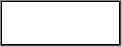
VISUALIZATION VISU_SubSystemButton  // 122x47
VAR_IN_OUT
    widget : SubSystemButtonWidget;
END_VAR
    Rectangle (0,0 120x45), invisible if: widget.isNotOrange
    Rectangle (0,0 120x45), invisible if: widget.isNotGray
    Rectangle (0,0 120x45), invisible if: widget.isNotBlue
    Rectangle (0,0 120x45), invisible if: widget.isNotRed
    Rectangle (0,0 120x45), invisible if: widget.isNotGreen
    Rectangle (0,0 120x45), "%s", text variable: widget.name
    Rectangle (0,0 120x45), invisible if: widget.notActivated
    Line (0,44) (120,44), invisible if: widget.activated
    Line (119,0) (119,45), invisible if: widget.activated
    Line (118,0) (0,0), invisible if: widget.activated
    Line (0,45) (0,0), invisible if: widget.activated
    Line (120,45) (120,1), invisible if: widget.notActivated
    Line (0,1) (119,1), invisible if: widget.notActivated
    Line (1,0) (1,45), invisible if: widget.notActivated
    Line (120,45) (1,45), invisible if: widget.notActivated
END_VISUALIZATION

(* stored: Version 1.1.0.1, ProductVersion 3.1.4019.2
   Visu VISU_SubSystemButton: Id {51a48865-cf23-400c-992d-6f921cfb6fa3} *)
